// TIA Portal V19 export
DATA_BLOCK "CallEquipment_DB"   // DB65
AUTHOR : Siemens_FA_SUP
// stored: InstanceOfName Unit2.Em5.CallEquipment, InstanceOfType FB, Namespace Unit2.Em5
"Unit2.Em5.CallEquipment"
   // VAR_IN_OUT
   //    unitStatus : "LAF_typeUnitStatus";
   //    unitAlarmDB : "LAF_typeAlarms";
   //    emFeedback : "LUC_typeEmFeedback";
   // END_VAR
   // VAR
   //    statUnitStatus { ExternalWritable := 'False'} : "LAF_typeUnitStatus";
   //    instJobExecute { ExternalWritable := 'False'} : "LAF_SelectJob";
   //    instJobStopping { ExternalWritable := 'False'; S7_SetPoint := 'True'} : "LAF_SelectJob";
   //    instJobStarting { ExternalWritable := 'False'; S7_SetPoint := 'True'} : "LAF_SelectJob";
   //    instJobHolding { ExternalWritable := 'False'; S7_SetPoint := 'True'} : "LAF_SelectJob";
   //    instJobUnHolding { ExternalWritable := 'False'; S7_SetPoint := 'True'} : "LAF_SelectJob";
   //    instJobRecover { ExternalWritable := 'False'; S7_SetPoint := 'True'} : "LAF_SelectJob";
   //    instJobReseting { ExternalWritable := 'False'; S7_SetPoint := 'True'} : "LAF_SelectJob";
   //    instSequence { ExternalWritable := 'False'} : "Unit2.Em5.Sequence";
   //    instManageBitAlarms { ExternalWritable := 'False'} : "LAF_ManageBitAlarms";
   //    instCmReset { ExternalWritable := 'False'; S7_SetPoint := 'True'} : "Unit2.Em5.EXCHANGETRAY_PlasticWorkstationCmResetOperator";
   //    instCm3SignalTM { ExternalWritable := 'False'} : "LEXCHANGETRAY_U2Em5SignalTM";
   //    instCm1Vfd208 { ExternalWritable := 'False'} : "LEXCHANGETRAY_RollerVfd";
   //    instCm2Cylinder { ExternalWritable := 'False'; S7_SetPoint := 'True'} : "LEXCHANGETRAY_Cylinder";
   //    instCm4SR1000Profinet { ExternalWritable := 'False'; S7_SetPoint := 'True'} : "LEXCHANGETRAY_Sr1000_Profinet";
   //    statLstUnitMode { ExternalWritable := 'False'; S7_SetPoint := 'True'} : DInt;   // 71
   // END_VAR
BEGIN
END_DATA_BLOCK
